{attribute 'enable_dynamic_creation'}
FUNCTION_BLOCK FB_ObjCollectionNode
VAR_INPUT
	pPrev : POINTER TO FB_ObjCollectionNode;
	pNext : POINTER TO FB_ObjCollectionNode;
END_VAR
VAR_OUTPUT
	nodes : FB_ObjCollection(THIS);
	pOwnerColl : POINTER TO FB_ObjCollection;
END_VAR
VAR
	pObject : POINTER TO FB_Object;
END_VAR

//Ist ein einzelnes Item einer Collection
//hat einen Vorgänger, Nachfolger, Parent(Collection), Nodes(Collection)

PROPERTY P_pOwnerColl : POINTER TO FB_ObjCollection
SET
pOwnerColl := P_pOwnerColl;
END_SET
GET
P_pOwnerColl := pOwnerColl;
END_GET
END_PROPERTY

PROPERTY P_pObject : POINTER TO FB_Object
GET
P_pObject := pObject;
END_GET
SET
pObject := P_pObject;
END_SET
END_PROPERTY

METHOD FB_init : BOOL
VAR_INPUT
	bInitRetains : BOOL; // if TRUE, the retain variables are initialized (warm start / cold start)
	bInCopyCode : BOOL;  // if TRUE, the instance afterwards gets moved into the copy code (online change)
	pOwnerColl : POINTER TO FB_ObjCollection;
END_VAR
THIS^.pOwnerColl := pOwnerColl;
END_METHOD

METHOD M_GetLevel : UINT
VAR_INPUT
	nStartLevel : UINT;
END_VAR
IF pOwnerColl^.pOwnerNode > 0 THEN
	nStartLevel := nStartLevel + 1;
	M_GetLevel := pOwnerColl^.pOwnerNode^.M_GetLevel(nStartLevel);
ELSE
	M_GetLevel := nStartLevel;
END_IF
END_METHOD

END_FUNCTION_BLOCK

(* stored: Version 1.1.0.1, ProductVersion 3.1.4020.12
   POU FB_ObjCollectionNode: Id {2bc56e7d-6c07-4680-9002-db755e53a932}, SpecialFunc None
   Property P_pOwnerColl: Id {3190258e-a26e-4ebb-bae9-3937e49ae072}
   Set Set: Id {890aadd1-58b7-4028-9a09-0ebbb838109f}
   Get Get: Id {b169cfca-f17e-4a81-978a-18dd6df75813}
   Property P_pObject: Id {80e466ae-88ce-4c9e-b796-bff6ff1c21a6}
   Get Get: Id {2d2308b8-a976-4ca9-b742-8e8760b155d8}
   Set Set: Id {8d93fdd4-5a3f-46b4-8b76-242edce93df7}
   Method FB_init: Id {af2586f4-5f95-4e36-b2b1-11c379b61c18}
   Method M_GetLevel: Id {e8dfeabe-9490-4db1-8f7b-8a7fa471b5bb} *)
